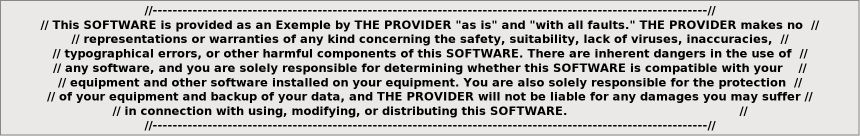
VISUALIZATION FrameDislaimer  // 860x136
    Rectangle (0,0 860x136), "//---------------------------------------------------------------------------------------------------------------// // This SOFTWARE is provided as an Exemple by THE PROVIDER "as is" and "with all faults." THE PROVIDER makes no // // representations or warranties of any kind concerning the safety, suitability, lack of viruses, inaccuracies, // // typographical errors, or other harmful components of this SOFTWARE. There are inherent dangers in the use of // // any software, and you are solely responsible for determining whether this SOFTWARE is compatible with your // // equipment and other software installed on your equipment. You are also solely responsible for the protection // // of your equipment and backup of your data, and THE PROVIDER will not be liable for any damages you may suffer // // in connection with using, modifying, or distributing this SOFTWARE. // //---------------------------------------------------------------------------------------------------------------//"
END_VISUALIZATION

(* stored: Version 1.1.0.1, ProductVersion 3.1.4024.12
   Visu FrameDislaimer: Id {2446d496-1816-4e06-8436-5be5491b1ba6} *)
